PROGRAM MAIN
VAR
	bLamp : BOOL;
	toggle: TON;
	toggleOff: TOF;
END_VAR

toggle(IN:= TRUE, PT:= T#2S , Q=>bLamp , ET=> );
toggleOff(IN:=TRUE , PT:=T#2S , Q=>bLamp , ET=> );

END_PROGRAM

(* stored: Version 1.1.0.1, ProductVersion 3.1.4024.12
   POU MAIN: Id {4d2f82b4-e367-4921-afc8-7510fc6e6aa2}, SpecialFunc None *)
